RoboDK station: Stringer C-Top2-BOX1.rdk

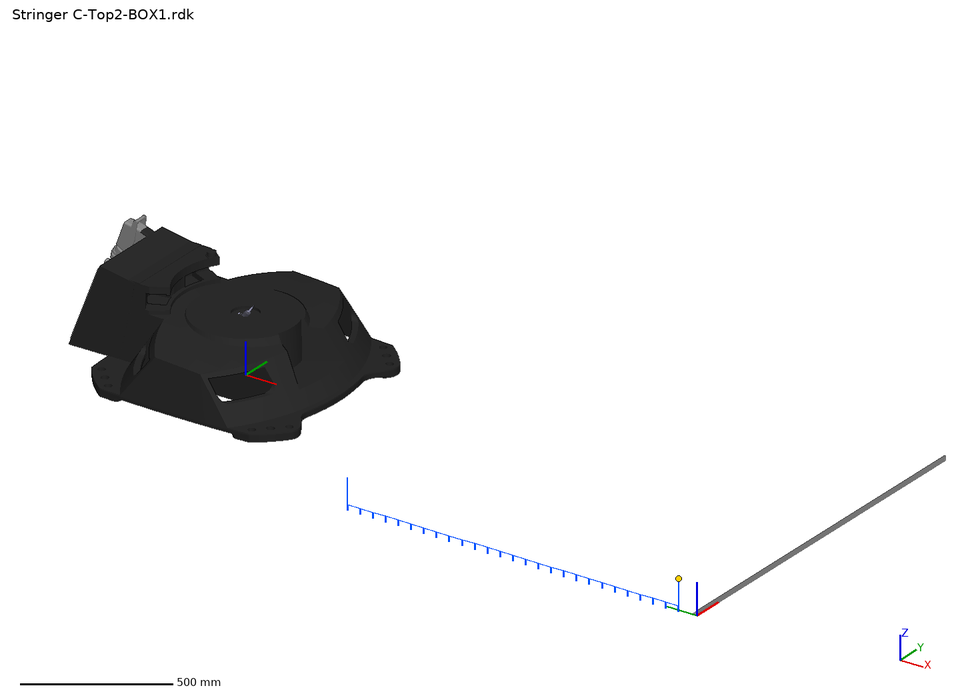
[picture v0: the station drawn from its stored meshes, robots at their saved joint values, targets as dots, program paths as lines]
Station Stringer C-Top2-BOX1 (saved by RoboDK 5.2.3). Poses are relative to the parent item; angles as X-Y-Z fixed-axis rotations.
  - frame KUKA KR 210 R2700 extra Base at (0, 0, 0) mm
    - robot KUKA KR 210 R2700 extra: 6 axes, payload 210 kg, reach 2696 mm, repeatability 0.06 mm, weight 1068 kg
        joint limits [-185, -140, -120, -350, -125, -350] to [185, -5, 155, 350, 125, 350]; home [0, -90, 90, 0, 0, 0]; saved at [-20.762, -27.449, 103.504, 149.833, 26.355, -168.904]
      - tool Spindle, TCP at (32, 0, 260) mm, rotated rx 0 ry 39 rz 0 deg, size 157.3 x 72 x 259.9 mm
  - frame Frame 2 at (1800, 0, -372.68) mm, rotated rx 0 ry 0 rz 90 deg
    - object L-Stringer C - Top2-BOX1 at (0, 0, 0) mm, size 1411.8 x 20 x 20 mm, geometry from L-Stringer C - Top2-BOX1.stl
    - object Stringer C-Top2-BOX1 at (0, 0, 0) mm, rotated rx 0 ry 0 rz -90 deg, 27 curves, geometry from Point 27
  - machining project Print3D settings: rotZ(0) | rotX(0)*rotY(0) | rotz(0) | onStart | onPathStart | onApproach | onPoint | onRetract | onFinish | SetRPM(%1) | SetTool(%1) | Extruder(%1) | default | default | OutOnMov(%1) | OutOffMov(%1) | onPathFinish | M_RunCode(%1)
  - program Print3D (146 instructions, listed below)
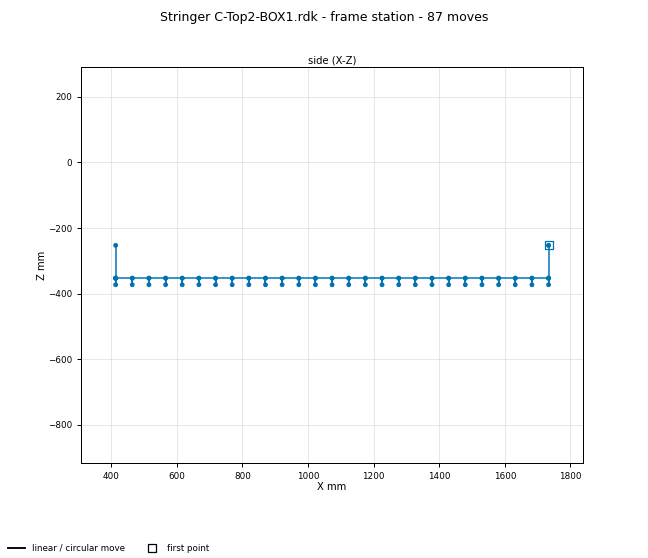
[picture p0: tool path of Stringer C-Top2-BOX1.rdk in frame station, 87 of 87 moves have a stored position in this frame; points joined in program order, loops and branches not executed]

--- program Print3D (robot KUKA KR 210 R2700 extra) ---
  Smooth(1)
  Set speed (1000.0 mm/s)
  Set Ref.: Frame 2
  Set Tool: Spindle
  Show Spindle
  MoveJ 1 to (-11.2, 66.57, 120) mm, rotated rx 180 ry 0 rz -180 deg; joints [-2.516, -34.012, 111.84, 176.492, 26.844, -178.825]
  MoveL 2 to (-11.2, 66.57, 120) mm, rotated rx 180 ry 0 rz -180 deg; joints [-2.516, -34.012, 111.84, 176.492, 26.844, -178.825]
  MoveL 3 to (-11.2, 66.57, 20) mm, rotated rx 180 ry 0 rz 180 deg; joints [-2.516, -28.683, 109.197, 176.786, 29.526, -179.159]
  MoveL 4 to (-11.2, 66.57, 20) mm, rotated rx 180 ry 0 rz 180 deg; joints [-2.516, -28.683, 109.197, 176.786, 29.526, -179.159]
  Set speed (50.0 mm/s)
  MoveL 5 to (-11.2, 66.57, 0) mm, rotated rx 180 ry 0 rz 180 deg; joints [-2.516, -27.625, 108.621, 176.833, 30.007, -179.213]
  MoveL 6 to (-11.2, 66.57, 20) mm, rotated rx 180 ry 0 rz 180 deg; joints [-2.516, -28.683, 109.197, 176.786, 29.526, -179.159]
  Set speed (1000.0 mm/s)
  MoveL 7 to (-11.2, 117.34, 20) mm, rotated rx -180 ry 0 rz -180 deg; joints [-4.43, -28.661, 109.037, 174.32, 29.413, -178.493]
  Set speed (50.0 mm/s)
  MoveL 8 to (-11.2, 117.34, 0) mm, rotated rx -180 ry 0 rz -180 deg; joints [-4.43, -27.605, 108.462, 174.403, 29.892, -178.589]
  MoveL 9 to (-11.2, 117.34, 20) mm, rotated rx -180 ry 0 rz -180 deg; joints [-4.43, -28.661, 109.037, 174.32, 29.413, -178.493]
  Set speed (1000.0 mm/s)
  MoveL 10 to (-11.2, 168.11, 20) mm, rotated rx -180 ry 0 rz -180 deg; joints [-6.333, -28.627, 108.79, 171.83, 29.24, -177.789]
  Set speed (50.0 mm/s)
  MoveL 11 to (-11.2, 168.11, 0) mm, rotated rx -180 ry 0 rz -180 deg; joints [-6.333, -27.572, 108.215, 171.95, 29.715, -177.927]
  MoveL 12 to (-11.2, 168.11, 20) mm, rotated rx -180 ry 0 rz -180 deg; joints [-6.333, -28.627, 108.79, 171.83, 29.24, -177.789]
  Set speed (1000.0 mm/s)
  MoveL 13 to (-11.2, 218.88, 20) mm, rotated rx -180 ry 0 rz -180 deg; joints [-8.222, -28.579, 108.454, 169.305, 29.01, -177.028]
  Set speed (50.0 mm/s)
  MoveL 14 to (-11.2, 218.88, 0) mm, rotated rx -180 ry 0 rz -180 deg; joints [-8.222, -27.528, 107.881, 169.462, 29.48, -177.209]
  MoveL 15 to (-11.2, 218.88, 20) mm, rotated rx -180 ry 0 rz -180 deg; joints [-8.222, -28.579, 108.454, 169.305, 29.01, -177.028]
  Set speed (1000.0 mm/s)
  MoveL 16 to (-11.2, 269.65, 20) mm, rotated rx -180 ry 0 rz -180 deg; joints [-10.094, -28.516, 108.031, 166.733, 28.726, -176.195]
  Set speed (50.0 mm/s)
  MoveL 17 to (-11.2, 269.65, 0) mm, rotated rx 180 ry 0 rz 180 deg; joints [-10.094, -27.469, 107.459, 166.929, 29.19, -176.419]
  MoveL 18 to (-11.2, 269.65, 20) mm, rotated rx -180 ry 0 rz -180 deg; joints [-10.094, -28.516, 108.031, 166.733, 28.726, -176.195]
  Set speed (1000.0 mm/s)
  MoveL 19 to (-11.2, 320.42, 20) mm, rotated rx -180 ry 0 rz -180 deg; joints [-11.944, -28.438, 107.52, 164.105, 28.394, -175.272]
  Set speed (50.0 mm/s)
  MoveL 20 to (-11.2, 320.42, 0) mm, rotated rx -180 ry 0 rz -180 deg; joints [-11.944, -27.395, 106.95, 164.34, 28.85, -175.54]
  MoveL 21 to (-11.2, 320.42, 20) mm, rotated rx -180 ry 0 rz -180 deg; joints [-11.944, -28.438, 107.52, 164.105, 28.394, -175.272]
  Set speed (1000.0 mm/s)
  MoveL 22 to (-11.2, 371.19, 20) mm, rotated rx -180 ry 0 rz -180 deg; joints [-13.769, -28.343, 106.923, 161.407, 28.02, -174.242]
  Set speed (50.0 mm/s)
  MoveL 23 to (-11.2, 371.19, 0) mm, rotated rx -180 ry 0 rz -180 deg; joints [-13.769, -27.305, 106.355, 161.684, 28.465, -174.557]
  MoveL 24 to (-11.2, 371.19, 20) mm, rotated rx -180 ry 0 rz -180 deg; joints [-13.769, -28.343, 106.923, 161.407, 28.02, -174.242]
  Set speed (1000.0 mm/s)
  MoveL 25 to (-11.2, 421.96, 20) mm, rotated rx 180 ry 0 rz 180 deg; joints [-15.566, -28.229, 106.238, 158.629, 27.609, -173.091]
  Set speed (50.0 mm/s)
  MoveL 26 to (-11.2, 421.96, 0) mm, rotated rx -180 ry 0 rz -180 deg; joints [-15.566, -27.197, 105.673, 158.948, 28.043, -173.452]
  MoveL 27 to (-11.2, 421.96, 20) mm, rotated rx 180 ry 0 rz 180 deg; joints [-15.566, -28.229, 106.238, 158.629, 27.609, -173.091]
  Set speed (1000.0 mm/s)
  MoveL 28 to (-11.2, 472.73, 20) mm, rotated rx 180 ry 0 rz -180 deg; joints [-17.332, -28.093, 105.468, 155.758, 27.169, -171.801]
  Set speed (50.0 mm/s)
  MoveL 29 to (-11.2, 472.73, 0) mm, rotated rx 180 ry 0 rz 180 deg; joints [-17.332, -27.068, 104.905, 156.122, 27.591, -172.211]
  MoveL 30 to (-11.2, 472.73, 20) mm, rotated rx 180 ry 0 rz -180 deg; joints [-17.332, -28.093, 105.468, 155.758, 27.169, -171.801]
  Set speed (1000.0 mm/s)
  MoveL 31 to (-11.2, 523.5, 20) mm, rotated rx 180 ry 0 rz -180 deg; joints [-19.065, -27.935, 104.611, 152.783, 26.709, -170.358]
  Set speed (50.0 mm/s)
  MoveL 32 to (-11.2, 523.5, 0) mm, rotated rx 180 ry 0 rz 180 deg; joints [-19.065, -26.917, 104.051, 153.192, 27.117, -170.818]
  MoveL 33 to (-11.2, 523.5, 20) mm, rotated rx 180 ry 0 rz -180 deg; joints [-19.065, -27.935, 104.611, 152.783, 26.709, -170.358]
  Set speed (1000.0 mm/s)
  MoveL 34 to (-11.2, 574.26, 20) mm, rotated rx 180 ry 0 rz 180 deg; joints [-20.762, -27.753, 103.669, 149.692, 26.236, -168.748]
  Set speed (50.0 mm/s)
  MoveL 35 to (-11.2, 574.26, 0) mm, rotated rx 180 ry 0 rz 180 deg; joints [-20.762, -26.742, 103.111, 150.149, 26.629, -169.258]
  MoveL 36 to (-11.2, 574.26, 20) mm, rotated rx 180 ry 0 rz 180 deg; joints [-20.762, -27.753, 103.669, 149.692, 26.236, -168.748]
  Set speed (1000.0 mm/s)
  MoveL 37 to (-11.2, 625.03, 20) mm, rotated rx 180 ry 0 rz 180 deg; joints [-22.423, -27.544, 102.642, 146.475, 25.762, -166.957]
  Set speed (50.0 mm/s)
  MoveL 38 to (-11.2, 625.03, 0) mm, rotated rx 180 ry 0 rz 180 deg; joints [-22.423, -26.54, 102.087, 146.98, 26.136, -167.518]
  MoveL 39 to (-11.2, 625.03, 20) mm, rotated rx 180 ry 0 rz 180 deg; joints [-22.423, -27.544, 102.642, 146.475, 25.762, -166.957]
  Set speed (1000.0 mm/s)
  MoveL 40 to (-11.2, 675.8, 20) mm, rotated rx 180 ry 0 rz -180 deg; joints [-24.044, -27.306, 101.529, 143.122, 25.294, -164.974]
  Set speed (50.0 mm/s)
  MoveL 41 to (-11.2, 675.8, 0) mm, rotated rx -180 ry 0 rz -180 deg; joints [-24.044, -26.311, 100.977, 143.675, 25.649, -165.587]
  MoveL 42 to (-11.2, 675.8, 20) mm, rotated rx 180 ry 0 rz -180 deg; joints [-24.044, -27.306, 101.529, 143.122, 25.294, -164.974]
  Set speed (1000.0 mm/s)
  MoveL 43 to (-11.2, 726.57, 20) mm, rotated rx -180 ry 0 rz -180 deg; joints [-25.625, -27.037, 100.332, 139.626, 24.845, -162.79]
  Set speed (50.0 mm/s)
  MoveL 44 to (-11.2, 726.57, 0) mm, rotated rx 180 ry 0 rz 180 deg; joints [-25.625, -26.05, 99.782, 140.227, 25.178, -163.454]
  MoveL 45 to (-11.2, 726.57, 20) mm, rotated rx -180 ry 0 rz -180 deg; joints [-25.625, -27.037, 100.332, 139.626, 24.845, -162.79]
  Set speed (1000.0 mm/s)
  MoveL 46 to (-11.2, 777.34, 20) mm, rotated rx 180 ry 0 rz -180 deg; joints [-27.166, -26.735, 99.049, 135.981, 24.424, -160.4]
  Set speed (50.0 mm/s)
  MoveL 47 to (-11.2, 777.34, 0) mm, rotated rx -180 ry 0 rz -180 deg; joints [-27.166, -25.758, 98.501, 136.63, 24.735, -161.113]
  MoveL 48 to (-11.2, 777.34, 20) mm, rotated rx 180 ry 0 rz -180 deg; joints [-27.166, -26.735, 99.049, 135.981, 24.424, -160.4]
  Set speed (1000.0 mm/s)
  MoveL 49 to (-11.2, 828.11, 20) mm, rotated rx -180 ry 0 rz -180 deg; joints [-28.665, -26.398, 97.681, 132.187, 24.043, -157.801]
  Set speed (50.0 mm/s)
  MoveL 50 to (-11.2, 828.11, 0) mm, rotated rx -180 ry 0 rz -180 deg; joints [-28.665, -25.43, 97.136, 132.88, 24.329, -158.562]
  MoveL 51 to (-11.2, 828.11, 20) mm, rotated rx -180 ry 0 rz -180 deg; joints [-28.665, -26.398, 97.681, 132.187, 24.043, -157.801]
  Set speed (1000.0 mm/s)
  MoveL 52 to (-11.2, 878.88, 20) mm, rotated rx 180 ry 0 rz 180 deg; joints [-30.123, -26.024, 96.227, 128.247, 23.713, -154.997]
  Set speed (50.0 mm/s)
  MoveL 53 to (-11.2, 878.88, 0) mm, rotated rx -180 ry 0 rz -180 deg; joints [-30.123, -25.066, 95.684, 128.981, 23.972, -155.8]
  MoveL 54 to (-11.2, 878.88, 20) mm, rotated rx 180 ry 0 rz 180 deg; joints [-30.123, -26.024, 96.227, 128.247, 23.713, -154.997]
  Set speed (1000.0 mm/s)
  MoveL 55 to (-11.2, 929.65, 20) mm, rotated rx 180 ry 0 rz 180 deg; joints [-31.539, -25.612, 94.687, 124.168, 23.444, -151.996]
  Set speed (50.0 mm/s)
  MoveL 56 to (-11.2, 929.65, 0) mm, rotated rx -180 ry 0 rz -180 deg; joints [-31.539, -24.662, 94.146, 124.939, 23.676, -152.836]
  MoveL 57 to (-11.2, 929.65, 20) mm, rotated rx 180 ry 0 rz 180 deg; joints [-31.539, -25.612, 94.687, 124.168, 23.444, -151.996]
  Set speed (1000.0 mm/s)
  MoveL 58 to (-11.2, 980.42, 20) mm, rotated rx -180 ry 0 rz -180 deg; joints [-32.913, -25.158, 93.06, 119.966, 23.248, -148.811]
  Set speed (50.0 mm/s)
  MoveL 59 to (-11.2, 980.42, 0) mm, rotated rx 180 ry 0 rz 180 deg; joints [-32.913, -24.218, 92.52, 120.765, 23.45, -149.682]
  MoveL 60 to (-11.2, 980.42, 20) mm, rotated rx -180 ry 0 rz -180 deg; joints [-32.913, -25.158, 93.06, 119.966, 23.248, -148.811]
  Set speed (1000.0 mm/s)
  MoveL 61 to (-11.2, 1031.19, 20) mm, rotated rx 180 ry 0 rz -180 deg; joints [-34.246, -24.661, 91.344, 115.66, 23.135, -145.465]
  Set speed (50.0 mm/s)
  MoveL 62 to (-11.2, 1031.19, 0) mm, rotated rx -180 ry 0 rz -180 deg; joints [-34.246, -23.73, 90.806, 116.48, 23.307, -146.357]
  MoveL 63 to (-11.2, 1031.19, 20) mm, rotated rx 180 ry 0 rz -180 deg; joints [-34.246, -24.661, 91.344, 115.66, 23.135, -145.465]
  Set speed (1000.0 mm/s)
  MoveL 64 to (-11.2, 1081.96, 20) mm, rotated rx -180 ry 0 rz -180 deg; joints [-35.538, -24.118, 89.539, 111.276, 23.113, -141.982]
  Set speed (50.0 mm/s)
  MoveL 65 to (-11.2, 1081.96, 0) mm, rotated rx -180 ry 0 rz -180 deg; joints [-35.538, -23.197, 89.001, 112.107, 23.254, -142.886]
  MoveL 66 to (-11.2, 1081.96, 20) mm, rotated rx -180 ry 0 rz -180 deg; joints [-35.538, -24.118, 89.539, 111.276, 23.113, -141.982]
  Set speed (1000.0 mm/s)
  MoveL 67 to (-11.2, 1132.73, 20) mm, rotated rx -180 ry 0 rz -180 deg; joints [-36.789, -23.528, 87.641, 106.844, 23.19, -138.394]
  Set speed (50.0 mm/s)
  MoveL 68 to (-11.2, 1132.73, 0) mm, rotated rx -180 ry 0 rz -180 deg; joints [-36.789, -22.616, 87.103, 107.676, 23.301, -139.299]
  MoveL 69 to (-11.2, 1132.73, 20) mm, rotated rx -180 ry 0 rz -180 deg; joints [-36.789, -23.528, 87.641, 106.844, 23.19, -138.394]
  Set speed (1000.0 mm/s)
  MoveL 70 to (-11.2, 1183.5, 20) mm, rotated rx 180 ry 0 rz 180 deg; joints [-38.001, -22.889, 85.648, 102.4, 23.373, -134.735]
  Set speed (50.0 mm/s)
  MoveL 71 to (-11.2, 1183.5, 0) mm, rotated rx 180 ry 0 rz -180 deg; joints [-38.001, -21.985, 85.11, 103.221, 23.454, -135.63]
  MoveL 72 to (-11.2, 1183.5, 20) mm, rotated rx 180 ry 0 rz 180 deg; joints [-38.001, -22.889, 85.648, 102.4, 23.373, -134.735]
  Set speed (1000.0 mm/s)
  MoveL 73 to (-11.2, 1234.26, 20) mm, rotated rx -180 ry 0 rz -180 deg; joints [-39.174, -22.196, 83.558, 97.978, 23.667, -131.044]
  Set speed (50.0 mm/s)
  MoveL 74 to (-11.2, 1234.26, 0) mm, rotated rx 180 ry 0 rz 180 deg; joints [-39.174, -21.301, 83.018, 98.778, 23.718, -131.917]
  MoveL 75 to (-11.2, 1234.26, 20) mm, rotated rx -180 ry 0 rz -180 deg; joints [-39.174, -22.196, 83.558, 97.978, 23.667, -131.044]
  Set speed (1000.0 mm/s)
  MoveL 76 to (-11.2, 1285.03, 20) mm, rotated rx 180 ry 0 rz 180 deg; joints [-40.31, -21.448, 81.365, 93.613, 24.075, -127.352]
  Set speed (50.0 mm/s)
  MoveL 77 to (-11.2, 1285.03, 0) mm, rotated rx -180 ry 0 rz -180 deg; joints [-40.31, -20.562, 80.823, 94.382, 24.099, -128.195]
  MoveL 78 to (-11.2, 1285.03, 20) mm, rotated rx 180 ry 0 rz 180 deg; joints [-40.31, -21.448, 81.365, 93.613, 24.075, -127.352]
  Set speed (1000.0 mm/s)
  MoveL 79 to (-11.2, 1335.8, 20) mm, rotated rx -180 ry 0 rz -180 deg; joints [-41.408, -20.642, 79.065, 89.336, 24.599, -123.695]
  Set speed (50.0 mm/s)
  MoveL 80 to (-11.2, 1335.8, 0) mm, rotated rx -180 ry 0 rz -180 deg; joints [-41.408, -19.763, 78.52, 90.066, 24.598, -124.497]
  MoveL 81 to (-11.2, 1335.8, 20) mm, rotated rx -180 ry 0 rz -180 deg; joints [-41.408, -20.642, 79.065, 89.336, 24.599, -123.695]
  Set speed (1000.0 mm/s)
  MoveL 82 to (-11.2, 1386.57, 20) mm, rotated rx 180 ry 0 rz -180 deg; joints [-42.47, -19.773, 76.652, 85.177, 25.241, -120.099]
  Set speed (50.0 mm/s)
  MoveL 83 to (-11.2, 1386.57, 0) mm, rotated rx 180 ry 0 rz -180 deg; joints [-42.47, -18.901, 76.103, 85.86, 25.216, -120.853]
  MoveL 84 to (-11.2, 1386.57, 20) mm, rotated rx 180 ry 0 rz -180 deg; joints [-42.47, -19.773, 76.652, 85.177, 25.241, -120.099]
  MoveL 85 to (-11.2, 1386.57, 20) mm, rotated rx 180 ry 0 rz -180 deg; joints [-42.47, -19.773, 76.652, 85.177, 25.241, -120.099]
  Set speed (1000.0 mm/s)
  MoveL 86 to (-11.2, 1386.57, 20) mm, rotated rx 180 ry 0 rz -180 deg; joints [-42.47, -19.773, 76.652, 85.177, 25.241, -120.099]
  MoveL 87 to (-11.2, 1386.57, 120) mm, rotated rx -180 ry 0 rz -180 deg; joints [-42.47, -24.063, 79.133, 81.383, 25.453, -115.9]
